(* IEC 61131-3 sources: plc_digit/, 2 files *)

(* ---- ff_jk.ST ---- *)
FUNCTION_BLOCK ff_jk
VAR_EXTERNAL

END_VAR

VAR_INPUT
my_ff_j	: bool;
my_ff_k	: bool;
my_clk : bool r_edge;
END_VAR

VAR_OUTPUT
my_ff_q	: bool;
END_VAR

VAR

END_VAR
if (my_clk) then
if (my_ff_j & my_ff_k) then
	my_ff_q := not my_ff_q;				(* Toggle *)
else if (not my_ff_j & my_ff_k) then
	my_ff_q := false;					(* Reset *)
else if (my_ff_j & not my_ff_k) then
	my_ff_q := true;					(* Set *)
end_if;
end_if;
end_if;
end_if;

END_FUNCTION_BLOCK

(* ---- timer.ST ---- *)
FUNCTION_BLOCK timer
VAR_EXTERNAL

END_VAR

VAR_INPUT
period : time;
END_VAR

VAR_OUTPUT
	output : bool;
END_VAR

VAR
	clock : TON;
END_VAR

clock(IN := true, PT := period);

if (clock.q) then
	output := not output;
	clock (in:= false);
end_if;

END_FUNCTION_BLOCK
